TYPE ST_AlarmSensorHMI :
STRUCT
	sName		: STRING;	// Sensor name
	nID			: INT;		// Alarm component ID
	bAlarm		: BOOL;		// True if the sensor detects something
	bTamper		: BOOL;		// True if the sensor is tampered with
	bDisabled	: BOOL;		// True if the sensor is disabled
END_STRUCT
END_TYPE

(* stored: Version 1.1.0.1, ProductVersion 3.1.4024.12
   DUT ST_AlarmSensorHMI: Id {af77090b-9d40-4dff-8455-e4047ab87e8f} *)
